Fanuc KAREL source: NC0078.KL

-- PROVISIONAL review KL for V940-1; original PC SHA256 162c861489e6d21fd943ac0a91cfbace4b740825ae3fbf19ed5b1af11802ffbb
-- Incomplete behavior may be omitted. Consult companion uncertainty JSON. Do not deploy.
PROGRAM NC0078
%NOLOCKGROUP
-- UNRESOLVED_LOCAL_POOL 1 cells at code offset 3; source declarations unknown
-- DIRECT_LOCAL_WORD_ACCESS alone does not prove INTEGER, REAL, or BOOLEAN
BEGIN
  -- V9_OWNER_INTERVAL_HINT [6,95),[11,93),[16,91),[21,89),[26,87),[31,85),[36,83),[41,81),[46,79),[51,77),[56,75),[61,73); structural only; source/VM held
  -- V9_EXPOSED_INDEXED_TABLE_HINT layout=0001; 24 counted words exposed once; source arms/runtime held
  -- UNRESOLVED_PC offsets 0-8; opcodes 2B,2C,7B
  -- UNRESOLVED_PC offsets 13-20; opcodes 9D,23
  -- UNRESOLVED_PC offsets 25-42; opcodes 21,2E,59,79
  -- UNRESOLVED_PC offsets 47-64; opcodes 21,2E,59,79
  -- UNRESOLVED_PC offsets 69-86; opcodes 21,2E,59,79
  -- UNRESOLVED_PC offsets 91-108; opcodes 21,2E,59,79
  -- UNRESOLVED_PC offsets 113-130; opcodes 21,2E,59,79
  -- UNRESOLVED_PC offsets 135-152; opcodes 21,2E,59,79
  -- UNRESOLVED_PC offsets 157-174; opcodes 21,2E,59,79
  -- UNRESOLVED_PC offsets 179-196; opcodes 21,2E,59,79
  -- UNRESOLVED_PC offsets 201-218; opcodes 21,2E,59,79
  -- UNRESOLVED_PC offsets 223-240; opcodes 21,2E,59,79
  -- UNRESOLVED_PC offsets 245-262; opcodes 21,2E,59,79
  -- UNRESOLVED_PC offsets 267-284; opcodes 21,2E,59,79
  -- UNRESOLVED_PC offsets 289-303; opcodes 21,9D,52,23
  -- UNRESOLVED_PC offsets 308-313; opcodes 7A
  -- UNRESOLVED_PC offsets 318-323; opcodes 7A
  -- UNRESOLVED_PC offsets 328-333; opcodes 7A
  -- UNRESOLVED_PC offsets 338-343; opcodes 7A
  -- UNRESOLVED_PC offsets 348-353; opcodes 7A
  -- UNRESOLVED_PC offsets 358-363; opcodes 7A
  -- UNRESOLVED_PC offsets 368-373; opcodes 7A
  -- UNRESOLVED_PC offsets 378-383; opcodes 7A
  -- UNRESOLVED_PC offsets 388-393; opcodes 7A
  -- UNRESOLVED_PC offsets 398-403; opcodes 7A
  -- UNRESOLVED_PC offsets 408-413; opcodes 7A
  -- UNRESOLVED_PC offsets 418-423; opcodes 7A
  -- UNRESOLVED_PC offsets 428-432; opcodes 7F
  -- UNRESOLVED_PC offsets 437-441; opcodes 27,AA
  -- UNRESOLVED_PC offsets 446-450; opcodes 7F
END NC0078
